FUNCTION F_Scale : INT
VAR_INPUT
	Value:	INT;
END_VAR
VAR
END_VAR

F_Scale := TO_INT((255.0/32767.0) * TO_REAL(Value));

END_FUNCTION

(* stored: Version 1.1.0.1, ProductVersion 3.1.4024.11
   POU F_Scale: Id {2e72596d-47d0-4300-958d-56d309a78999}, SpecialFunc None *)
